(* IEC 61131-3 sources: CodesysTest/alpha/export/FBs/Components/LoadPlate/FB_BaseLoadPlate.pou/Shaking.prop, 1 file *)

(* ---- Get.pm.st ---- *)
(*#-#-#-#-#-#-#-#-#-#---Declaration---#-#-#-#-#-#-#-#-#-#-#-#-#*)

VAR
END_VAR
(*#-#-#-#-#-#-#-#-#-#---Implementation---#-#-#-#-#-#-#-#-#-#-#-#-#*)

Shaking := _shake OR _shaking;
